// TIA Portal V16 export
// export: Created 2024-04-19T15:29:40.8774347Z, ExportSetting WithDefaults, DisplayName Totally Integrated Automation Portal, DisplayVersion V16 Update 6, DisplayName TIA Portal Version Control Interface, DisplayVersion V16 Update 2, DisplayName TIA Portal Openness, DisplayVersion V16 Update 6, DisplayName TIA Portal Test Suite Advanced, DisplayVersion V16, DisplayName SINAMICS Startdrive Advanced, DisplayVersion V16 Update 5, DisplayName SINAMICS Startdrive G130, G150, S120, S150, SINAMICS MV, S210, DisplayVersion V16 Update 5, DisplayName SINAMICS Startdrive G110M, G120, G120C, G120D, G120P, G115D, DisplayVersion V16 Update 5, DisplayName STEP 7 Professional, DisplayVersion V16 Update 6, DisplayName STEP 7 Safety, DisplayVersion V16, DisplayName WinCC Advanced, DisplayVersion V16 Update 6
TYPE "SCA_rapidDoor_IO"
// stored: IsFailsafeCompliant false
   STRUCT
      Safety_switch : Bool;   // Safety switch
      Entry_pec : Bool;   // Entry photocell
      Exit_pec : Bool;   // Exit photocell
      Open : Bool;   // Door open
      Closed : Bool;   // Door closed
      Man_open : Bool;   // Open door manual switch
      Man_close : Bool;   // Close door manual switch
      Open_req : Bool;   // Output: Up request
      Close_req : Bool;   // Output: Down request
      Impulsdrift : Bool;   // Output: Impuls drift
   END_STRUCT;
END_TYPE
